// TIA Portal project "Event_Report" (V21)

(* hardware
DEVICE "S7-1200 station_1"  S7-1200 Station
   slot 0: "Rack_0"  S7-1200 Rack  Rack  V1.0
   slot 1: "PLC_1"  CPU 1215C AC/DC/Rly  6ES7 215-1BG40-0XB0  V4.2
*)

// ===== PLC "PLC_1"  CPU 1215C AC/DC/Rly =====

TYPE "UDT_CommBuffer"
VERSION : 0.1
   STRUCT
      SendTrigger : Bool;
      SendBuffer : Array[0..1023] of Byte;
      RecvBuffer : Array[0..1023] of Byte;
      RecvLength : UInt;
      RecvReady : Bool;
   END_STRUCT;
END_TYPE

DATA_BLOCK "DB_InputMonitor"   // DB1
{ S7_Optimized_Access := 'TRUE' }
VERSION : 0.1
   VAR
      InputImage : Array[1..100] of DWord;
      InputImage_Old : Array[1..100] of DWord;
      bSending : Bool;
   END_VAR
BEGIN
END_DATA_BLOCK

DATA_BLOCK "DB_CommData"   // DB3
{ S7_Optimized_Access := 'TRUE' }
AUTHOR : SIMATIC
VERSION : 0.1
   VAR
      SendLength : UInt;
      RecvLength : UInt;
      SendBuffer : Array[0..255] of Byte;
      RecvBuffer : Array[0..255] of Byte;
      StatusWord : Word;
   END_VAR
BEGIN
END_DATA_BLOCK

DATA_BLOCK "IDB_UdpTx"   // DB5
{ S7_Optimized_Access := 'TRUE' }
VERSION : 0.1
// stored: InstanceOfName FB_UdpTx
"FB_UdpTx"
BEGIN
END_DATA_BLOCK

DATA_BLOCK "IDB_MapDBtoIO"   // DB6
{ S7_Optimized_Access := 'TRUE' }
VERSION : 0.1
// stored: InstanceOfName FB_MapDBtoIO
"FB_MapDBtoIO"
BEGIN
   enable := true;
   tgtByte := 2;
   srcDB := 10;
   srcEndByte := 27;
   area := 16#81;
END_DATA_BLOCK

DATA_BLOCK "DB_input"   // DB10
{ S7_Optimized_Access := 'FALSE' }
VERSION : 0.1
   VAR
      "1层上行召梯按钮" : Bool;
      "2层上行召梯按钮" : Bool;
      "3层上行召梯按钮" : Bool;
      "4层上行召梯按钮" : Bool;
      "5层上行召梯按钮" : Bool;
      "6层上行召梯按钮" : Bool;
      "7层上行召梯按钮" : Bool;
      "8层上行召梯按钮" : Bool;
      "9层上行召梯按钮" : Bool;
      "2层下行召梯按钮" : Bool;
      "3层下行召梯按钮" : Bool;
      "4层下行召梯按钮" : Bool;
      "5层下行召梯按钮" : Bool;
      "6层下行召梯按钮" : Bool;
      "7层下行召梯按钮" : Bool;
      "8层下行召梯按钮" : Bool;
      "9层下行召梯按钮" : Bool;
      "10层下行召梯按钮" : Bool;
      "1号桥轿内选层按钮1" : Bool;
      "1号桥轿内选层按钮2" : Bool;
      "1号桥轿内选层按钮3" : Bool;
      "1号桥轿内选层按钮4" : Bool;
      "1号桥轿内选层按钮5" : Bool;
      "1号桥轿内选层按钮6" : Bool;
      "1号桥轿内选层按钮7" : Bool;
      "1号桥轿内选层按钮8" : Bool;
      "1号桥轿内选层按钮9" : Bool;
      "1号桥轿内选层按钮10" : Bool;
      "1号桥轿内开门按钮" : Bool;
      "1号桥轿内关门按钮" : Bool;
      "1号桥光幕信号" : Bool;
      "1号桥超重信号" : Bool;
      "1号桥检修信号" : Bool;
      "1号桥轿厢门门锁信号" : Bool;
      "1号桥1楼层门门锁信号" : Bool;
      "1号桥2楼层门门锁信号" : Bool;
      "1号桥3楼层门门锁信号" : Bool;
      "1号桥4楼层门门锁信号" : Bool;
      "1号桥5楼层门门锁信号" : Bool;
      "1号桥6楼层门门锁信号" : Bool;
      "1号桥7楼层门门锁信号" : Bool;
      "1号桥8楼层门门锁信号" : Bool;
      "1号桥9楼层门门锁信号" : Bool;
      "1号桥10楼层门门锁信号" : Bool;
      "1号桥开门到位" : Bool;
      "1号桥关门到位" : Bool;
      "1号桥上平层信号" : Bool;
      "1号桥下平层信号" : Bool;
      "1号桥上端站第1限位" : Bool;
      "1号桥上端站第2限位" : Bool;
      "1号桥下端站第1限位" : Bool;
      "1号桥下端站第2限位" : Bool;
      "2号桥轿内选层按钮1" : Bool;
      "2号桥轿内选层按钮2" : Bool;
      "2号桥轿内选层按钮3" : Bool;
      "2号桥轿内选层按钮4" : Bool;
      "2号桥轿内选层按钮5" : Bool;
      "2号桥轿内选层按钮6" : Bool;
      "2号桥轿内选层按钮7" : Bool;
      "2号桥轿内选层按钮8" : Bool;
      "2号桥轿内选层按钮9" : Bool;
      "2号桥轿内选层按钮10" : Bool;
      "2号桥轿内开门按钮" : Bool;
      "2号桥轿内关门按钮" : Bool;
      "2号桥光幕信号" : Bool;
      "2号桥超重信号" : Bool;
      "2号桥检修信号" : Bool;
      "2号桥轿厢门门锁信号" : Bool;
      "2号桥1楼层门门锁信号" : Bool;
      "2号桥2楼层门门锁信号" : Bool;
      "2号桥3楼层门门锁信号" : Bool;
      "2号桥4楼层门门锁信号" : Bool;
      "2号桥5楼层门门锁信号" : Bool;
      "2号桥6楼层门门锁信号" : Bool;
      "2号桥7楼层门门锁信号" : Bool;
      "2号桥8楼层门门锁信号" : Bool;
      "2号桥9楼层门门锁信号" : Bool;
      "2号桥10楼层门门锁信号" : Bool;
      "2号桥开门到位" : Bool;
      "2号桥关门到位" : Bool;
      "2号桥上平层信号" : Bool;
      "2号桥下平层信号" : Bool;
      "2号桥上端站第1限位" : Bool;
      "2号桥上端站第2限位" : Bool;
      "2号桥下端站第1限位" : Bool;
      "2号桥下端站第2限位" : Bool;
      "3号桥轿内选层按钮1" : Bool;
      "3号桥轿内选层按钮2" : Bool;
      "3号桥轿内选层按钮3" : Bool;
      "3号桥轿内选层按钮4" : Bool;
      "3号桥轿内选层按钮5" : Bool;
      "3号桥轿内选层按钮6" : Bool;
      "3号桥轿内选层按钮7" : Bool;
      "3号桥轿内选层按钮8" : Bool;
      "3号桥轿内选层按钮9" : Bool;
      "3号桥轿内选层按钮10" : Bool;
      "3号桥轿内开门按钮" : Bool;
      "3号桥轿内关门按钮" : Bool;
      "3号桥光幕信号" : Bool;
      "3号桥超重信号" : Bool;
      "3号桥检修信号" : Bool;
      "3号桥轿厢门门锁信号" : Bool;
      "3号桥1楼层门门锁信号" : Bool;
      "3号桥2楼层门门锁信号" : Bool;
      "3号桥3楼层门门锁信号" : Bool;
      "3号桥4楼层门门锁信号" : Bool;
      "3号桥5楼层门门锁信号" : Bool;
      "3号桥6楼层门门锁信号" : Bool;
      "3号桥7楼层门门锁信号" : Bool;
      "3号桥8楼层门门锁信号" : Bool;
      "3号桥9楼层门门锁信号" : Bool;
      "3号桥10楼层门门锁信号" : Bool;
      "3号桥开门到位" : Bool;
      "3号桥关门到位" : Bool;
      "3号桥上平层信号" : Bool;
      "3号桥下平层信号" : Bool;
      "3号桥上端站第1限位" : Bool;
      "3号桥上端站第2限位" : Bool;
      "3号桥下端站第1限位" : Bool;
      "3号桥下端站第2限位" : Bool;
      "4号桥轿内选层按钮1" : Bool;
      "4号桥轿内选层按钮2" : Bool;
      "4号桥轿内选层按钮3" : Bool;
      "4号桥轿内选层按钮4" : Bool;
      "4号桥轿内选层按钮5" : Bool;
      "4号桥轿内选层按钮6" : Bool;
      "4号桥轿内选层按钮7" : Bool;
      "4号桥轿内选层按钮8" : Bool;
      "4号桥轿内选层按钮9" : Bool;
      "4号桥轿内选层按钮10" : Bool;
      "4号桥轿内开门按钮" : Bool;
      "4号桥轿内关门按钮" : Bool;
      "4号桥光幕信号" : Bool;
      "4号桥超重信号" : Bool;
      "4号桥检修信号" : Bool;
      "4号桥轿厢门门锁信号" : Bool;
      "4号桥1楼层门门锁信号" : Bool;
      "4号桥2楼层门门锁信号" : Bool;
      "4号桥3楼层门门锁信号" : Bool;
      "4号桥4楼层门门锁信号" : Bool;
      "4号桥5楼层门门锁信号" : Bool;
      "4号桥6楼层门门锁信号" : Bool;
      "4号桥7楼层门门锁信号" : Bool;
      "4号桥8楼层门门锁信号" : Bool;
      "4号桥9楼层门门锁信号" : Bool;
      "4号桥10楼层门门锁信号" : Bool;
      "4号桥开门到位" : Bool;
      "4号桥关门到位" : Bool;
      "4号桥上平层信号" : Bool;
      "4号桥下平层信号" : Bool;
      "4号桥上端站第1限位" : Bool;
      "4号桥上端站第2限位" : Bool;
      "4号桥下端站第1限位" : Bool;
      "4号桥下端站第2限位" : Bool;
      "5号桥轿内选层按钮1" : Bool;
      "5号桥轿内选层按钮2" : Bool;
      "5号桥轿内选层按钮3" : Bool;
      "5号桥轿内选层按钮4" : Bool;
      "5号桥轿内选层按钮5" : Bool;
      "5号桥轿内选层按钮6" : Bool;
      "5号桥轿内选层按钮7" : Bool;
      "5号桥轿内选层按钮8" : Bool;
      "5号桥轿内选层按钮9" : Bool;
      "5号桥轿内选层按钮10" : Bool;
      "5号桥轿内开门按钮" : Bool;
      "5号桥轿内关门按钮" : Bool;
      "5号桥光幕信号" : Bool;
      "5号桥超重信号" : Bool;
      "5号桥检修信号" : Bool;
      "5号桥轿厢门门锁信号" : Bool;
      "5号桥1楼层门门锁信号" : Bool;
      "5号桥2楼层门门锁信号" : Bool;
      "5号桥3楼层门门锁信号" : Bool;
      "5号桥4楼层门门锁信号" : Bool;
      "5号桥5楼层门门锁信号" : Bool;
      "5号桥6楼层门门锁信号" : Bool;
      "5号桥7楼层门门锁信号" : Bool;
      "5号桥8楼层门门锁信号" : Bool;
      "5号桥9楼层门门锁信号" : Bool;
      "5号桥10楼层门门锁信号" : Bool;
      "5号桥开门到位" : Bool;
      "5号桥关门到位" : Bool;
      "5号桥上平层信号" : Bool;
      "5号桥下平层信号" : Bool;
      "5号桥上端站第1限位" : Bool;
      "5号桥上端站第2限位" : Bool;
      "5号桥下端站第1限位" : Bool;
      "5号桥下端站第2限位" : Bool;
      "6号桥轿内选层按钮1" : Bool;
      "6号桥轿内选层按钮2" : Bool;
      "6号桥轿内选层按钮3" : Bool;
      "6号桥轿内选层按钮4" : Bool;
      "6号桥轿内选层按钮5" : Bool;
      "6号桥轿内选层按钮6" : Bool;
      "6号桥轿内选层按钮7" : Bool;
      "6号桥轿内选层按钮8" : Bool;
      "6号桥轿内选层按钮9" : Bool;
      "6号桥轿内选层按钮10" : Bool;
      "6号桥轿内开门按钮" : Bool;
      "6号桥轿内关门按钮" : Bool;
      "6号桥光幕信号" : Bool;
      "6号桥超重信号" : Bool;
      "6号桥检修信号" : Bool;
      "6号桥轿厢门门锁信号" : Bool;
      "6号桥1楼层门门锁信号" : Bool;
      "6号桥2楼层门门锁信号" : Bool;
      "6号桥3楼层门门锁信号" : Bool;
      "6号桥4楼层门门锁信号" : Bool;
      "6号桥5楼层门门锁信号" : Bool;
      "6号桥6楼层门门锁信号" : Bool;
      "6号桥7楼层门门锁信号" : Bool;
      "6号桥8楼层门门锁信号" : Bool;
      "6号桥9楼层门门锁信号" : Bool;
      "6号桥10楼层门门锁信号" : Bool;
      "6号桥开门到位" : Bool;
      "6号桥关门到位" : Bool;
      "6号桥上平层信号" : Bool;
      "6号桥下平层信号" : Bool;
      "6号桥上端站第1限位" : Bool;
      "6号桥上端站第2限位" : Bool;
      "6号桥下端站第1限位" : Bool;
      "6号桥下端站第2限位" : Bool;
      自动运行信号 : Bool;
   END_VAR
BEGIN
END_DATA_BLOCK

DATA_BLOCK "DB_output"   // DB11
{ S7_Optimized_Access := 'FALSE' }
VERSION : 0.1
   VAR
      "1" : Bool;
      "2" : Bool;
      "3" : Bool;
      "4" : Bool;
      "5" : Bool;
      "6" : Bool;
      "7" : Bool;
      "8" : Bool;
      "9" : Bool;
      "10" : Bool;
      "11" : Bool;
      "12" : Bool;
      "13" : Bool;
      "14" : Bool;
      "15" : Bool;
      "16" : Bool;
      "17" : Bool;
      "18" : Bool;
      "19" : Bool;
      "20" : Bool;
      "21" : Bool;
      "22" : Bool;
      "23" : Bool;
      "24" : Bool;
      "25" : Bool;
      "26" : Bool;
      "27" : Bool;
      "28" : Bool;
      "29" : Bool;
      "30" : Bool;
      "31" : Bool;
      "32" : Bool;
      "33" : Bool;
      "34" : Bool;
      "35" : Bool;
      "36" : Bool;
      "37" : Bool;
      "38" : Bool;
      "39" : Bool;
      "40" : Bool;
      "41" : Bool;
      "42" : Bool;
      "43" : Bool;
      "44" : Bool;
      "45" : Bool;
      "46" : Bool;
      "47" : Bool;
      "48" : Bool;
      "49" : Bool;
      "50" : Bool;
      "51" : Bool;
      "52" : Bool;
      "53" : Bool;
      "54" : Bool;
      "55" : Bool;
      "56" : Bool;
      "57" : Bool;
      "58" : Bool;
      "59" : Bool;
      "60" : Bool;
      "61" : Bool;
      "62" : Bool;
      "63" : Bool;
      "64" : Bool;
      "65" : Bool;
      "66" : Bool;
      "67" : Bool;
      "68" : Bool;
      "69" : Bool;
      "70" : Bool;
      "71" : Bool;
      "72" : Bool;
      "73" : Bool;
      "74" : Bool;
      "75" : Bool;
      "76" : Bool;
      "77" : Bool;
      "78" : Bool;
      "79" : Bool;
      "80" : Bool;
      "81" : Bool;
      "82" : Bool;
      "83" : Bool;
      "84" : Bool;
      "85" : Bool;
      "86" : Bool;
      "87" : Bool;
      "88" : Bool;
      "89" : Bool;
      "90" : Bool;
      "91" : Bool;
      "92" : Bool;
      "93" : Bool;
      "94" : Bool;
      "95" : Bool;
      "96" : Bool;
      "97" : Bool;
      "98" : Bool;
      "99" : Bool;
      "100" : Bool;
      "101" : Bool;
      "102" : Bool;
      "103" : Bool;
      "104" : Bool;
      "105" : Bool;
      "106" : Bool;
      "107" : Bool;
      "108" : Bool;
      "109" : Bool;
      "110" : Bool;
      "111" : Bool;
      "112" : Bool;
      "113" : Bool;
      "114" : Bool;
      "115" : Bool;
      "116" : Bool;
      "117" : Bool;
      "118" : Bool;
      "119" : Bool;
      "120" : Bool;
      "121" : Bool;
      "122" : Bool;
      "123" : Bool;
      "124" : Bool;
      "125" : Bool;
      "126" : Bool;
      "127" : Bool;
      "128" : Bool;
      "129" : Bool;
      "130" : Bool;
      "131" : Bool;
      "132" : Bool;
      "133" : Bool;
      "134" : Bool;
      "135" : Bool;
      "136" : Bool;
      "137" : Bool;
      "138" : Bool;
      "139" : Bool;
      "140" : Bool;
      "141" : Bool;
      "142" : Bool;
      "143" : Bool;
      "144" : Bool;
      "145" : Bool;
      "146" : Bool;
      "147" : Bool;
      "148" : Bool;
      "149" : Bool;
      "150" : Bool;
      "151" : Bool;
      "152" : Bool;
      "153" : Bool;
      "154" : Bool;
      "155" : Bool;
      "156" : Bool;
      "157" : Bool;
      "158" : Bool;
      "159" : Bool;
      "160" : Bool;
      "161" : Bool;
      "162" : Bool;
      "163" : Bool;
      "164" : Bool;
      "165" : Bool;
      "166" : Bool;
      "167" : Bool;
      "168" : Bool;
      "169" : Bool;
      "170" : Bool;
      "171" : Bool;
      "172" : Bool;
      "173" : Bool;
      "174" : Bool;
      "175" : Bool;
      "176" : Bool;
      "177" : Bool;
      "178" : Bool;
      "179" : Bool;
      "180" : Bool;
      "181" : Bool;
      "182" : Bool;
      "183" : Bool;
      "184" : Bool;
      "185" : Bool;
      "186" : Bool;
      "187" : Bool;
      "188" : Bool;
      "189" : Bool;
      "190" : Bool;
      "191" : Bool;
      "192" : Bool;
      "193" : Bool;
      "194" : Bool;
      "195" : Bool;
      "196" : Bool;
      "197" : Bool;
      "198" : Bool;
      "199" : Bool;
      "200" : Bool;
      "201" : Bool;
      "202" : Bool;
      "203" : Bool;
      "204" : Bool;
      "205" : Bool;
      "206" : Bool;
      "207" : Bool;
      "208" : Bool;
      "209" : Bool;
      "210" : Bool;
      "211" : Bool;
      "212" : Bool;
      "213" : Bool;
      "214" : Bool;
      "215" : Bool;
      "216" : Bool;
      "217" : Bool;
      "218" : Bool;
      "219" : Bool;
      "220" : Bool;
      "221" : Bool;
      "222" : Bool;
      "223" : Bool;
      "224" : Bool;
      "225" : Bool;
      "226" : Bool;
      "227" : Bool;
      "228" : Bool;
      "229" : Bool;
      "230" : Bool;
      "231" : Bool;
      "232" : Bool;
      "233" : Bool;
      "234" : Bool;
      "235" : Bool;
      "236" : Bool;
      "237" : Bool;
      "238" : Bool;
      "239" : Bool;
      "240" : Bool;
      "241" : Bool;
      "242" : Bool;
      "243" : Bool;
      "244" : Bool;
      "245" : Bool;
      "246" : Bool;
      "247" : Bool;
      "248" : Bool;
      "249" : Bool;
      "250" : Bool;
      "251" : Bool;
      "252" : Bool;
      "253" : Bool;
      "254" : Bool;
      "255" : Bool;
      "256" : Bool;
      "257" : Bool;
      "258" : Bool;
      "259" : Bool;
      "260" : Bool;
      "261" : Bool;
      "262" : Bool;
      "263" : Bool;
      "264" : Bool;
   END_VAR
BEGIN
END_DATA_BLOCK

// folder: System blocks/Program resources

DATA_BLOCK "DB_TCON_Param"   // DB2
{ S7_Optimized_Access := 'TRUE' }
AUTHOR : SIMATIC
FAMILY : MC7Plus
NAME : TCON_Prm
VERSION : 1.0
// stored: InstanceOfName TCON_Param
"TCON_Param"
BEGIN
   ID := 1;
   LOCAL_TSAP_ID_LEN := 2;
   LOCAL_TSAP_ID[1] := 16#07;
   LOCAL_TSAP_ID[2] := 16#D0;
   REM_STADDR[1] := 192;
   REM_STADDR[2] := 168;
   REM_STADDR[3] := 1;
   REM_STADDR[4] := 201;
   REM_TSAP_ID[1] := 16#2C;
   REM_TSAP_ID[2] := 16#BB;
   CONNECTION_TYPE := 19;
   ACTIVE_EST := false;
END_DATA_BLOCK

// folder: (top level)

FUNCTION_BLOCK "FB_MapDBtoIO"   // FB1, SCL
{ S7_Optimized_Access := 'TRUE' }
VERSION : 0.1
   VAR_OUTPUT
      mappedBytes : Int;
      targetEndByte : Int;
   END_VAR
   VAR
      enable : Bool;
      tgtByte : Int;
      tgtBit : Int;
      srcDB : Int;
      srcByte : Int;
      srcEndByte : Int;
      area : Int;
      areaDB : Int;
   END_VAR
   VAR_TEMP
      i : Int;
      totalBits : Int;
      "b" : Bool;
      curByte : Int;
      curBit : Int;
      tByte : Int;
      tBit : Int;
   END_VAR
BEGIN
   // 计算映射字节数与目标结束字节
   #mappedBytes := #srcEndByte - #srcByte + 1;
   #targetEndByte := #tgtByte + #mappedBytes - 1;
   IF #tgtBit > 0 THEN
       #targetEndByte := #targetEndByte + 1;
   END_IF;

   IF #enable THEN
       #totalBits := #mappedBytes * 8 - 1;
       FOR #i := 0 TO #totalBits DO
           #curByte := #srcByte + #i / 8;
           #curBit  := #i MOD 8;
           #b := PEEK_BOOL(area := 16#84, dbNumber := #srcDB, byteOffset := #curByte, bitOffset := #curBit);
           #tByte := #tgtByte + (#tgtBit + #i) / 8;
           #tBit  := (#tgtBit + #i) MOD 8;
           POKE_BOOL(area := #area, dbNumber := #areaDB, byteOffset := #tByte, bitOffset := #tBit, value := #b);
       END_FOR;
   END_IF;
END_FUNCTION_BLOCK

FUNCTION_BLOCK "FB_UdpTx"   // FB2, SCL
{ S7_Optimized_Access := 'TRUE' }
VERSION : 0.1
   VAR_INPUT
      SendData : Bool;
   END_VAR
   VAR_OUTPUT
      SendDone : Bool;
      SendBusy : Bool;
      SendError : Bool;
      SendStatus : Word;
      UdpReady : Bool;
   END_VAR
   VAR
      tconInst : TCON;
      tusendInst : TUSEND;
      tconEdge : Bool;
      tconMem : Bool;
      tusendEdge : Bool;
      tusendMem : Bool;
      tconDone : Bool;
      tconBusy : Bool;
      tconErr : Bool;
      tconStat : Word;
      tusendDone : Bool;
      tusendBusy : Bool;
      tusendErr : Bool;
      tusendStat : Word;
      udpBound : Bool;
      remoteAddr : TADDR_Param;
      addrInit : Bool;
   END_VAR
BEGIN
   // Init remote address once
   IF NOT #addrInit THEN
       #remoteAddr.REM_IP_ADDR[1] := 192;
       #remoteAddr.REM_IP_ADDR[2] := 168;
       #remoteAddr.REM_IP_ADDR[3] := 1;
       #remoteAddr.REM_IP_ADDR[4] := 201;
       #remoteAddr.REM_PORT_NR := 11451;
       #addrInit := TRUE;
   END_IF;

   // TCON: bind UDP socket
   #tconEdge := NOT #udpBound AND NOT #tconMem;
   #tconMem := NOT #udpBound;
   #tconInst(REQ := #tconEdge,
             ID := 1,
             CONNECT := "DB_TCON_Param",
             DONE => #tconDone,
             BUSY => #tconBusy,
             ERROR => #tconErr,
             STATUS => #tconStat);
   IF #tconDone THEN
       #udpBound := TRUE;
   END_IF;
   IF #tconErr THEN
       #tconMem := FALSE;
   END_IF;

   // TUSEND: fire and forget
   // InputImage[1..25] = 100 bytes, 保持原 LEN=100 兼容旧接收端
   #tusendEdge := #SendData AND #udpBound AND NOT #tusendMem;
   #tusendMem := #SendData;
   #tusendInst(REQ := #tusendEdge,
               ID := 1,
               LEN := 100,
               DATA := "DB_CommData".SendBuffer,
               ADDR := #remoteAddr,
               DONE => #tusendDone,
               BUSY => #tusendBusy,
               ERROR => #tusendErr,
               STATUS => #tusendStat);

   #SendDone := #tusendDone;
   #SendBusy := #tusendBusy;
   #SendError := #tusendErr;
   #SendStatus := #tusendStat;
   #UdpReady := #udpBound;
END_FUNCTION_BLOCK

ORGANIZATION_BLOCK "OB100"   // OB1, SCL, ProgramCycle
TITLE = "Main Program Sweep (Cycle)"
{ S7_Optimized_Access := 'TRUE' }
VERSION : 0.1
   VAR_INPUT
      Initial_Call : Bool;   // Initial call of this OB
      Remanence : Bool;   // =True, if remanent data are available
   END_VAR
   VAR_TEMP
      i : Int;
   END_VAR
BEGIN
   FOR #i := 1 TO 100 DO
       "DB_InputMonitor".InputImage[#i] := 0;
   END_FOR;
END_ORGANIZATION_BLOCK

ORGANIZATION_BLOCK "Main"   // OB1, SCL, ProgramCycle
TITLE = "Main Program Sweep (Cycle)"
{ S7_Optimized_Access := 'TRUE' }
VERSION : 0.1
   VAR_INPUT
      Initial_Call : Bool;   // Initial call of this OB
      Remanence : Bool;   // =True, if remanent data are available
   END_VAR
   VAR_TEMP
      i : Int;
      dwTemp : DWord;
      j : Int;
      idx : Int;
      dwInp : DWord;
      bChanged : Bool;
      mapBytes : Int;
      targetEndByte : Int;
      readStart : Int;
      readIdx : Int;
   END_VAR
BEGIN
   // 0: 动态映射 DB10 → I 区（参数在 IDB_MapDBtoIO 在线设置）
   "IDB_MapDBtoIO"();
   #mapBytes := "IDB_MapDBtoIO".mappedBytes;
   #targetEndByte := "IDB_MapDBtoIO".targetEndByte;

   // 1: 清零 InputImage
   FOR #i := 1 TO 25 DO
       "DB_InputMonitor".InputImage[#i] := 0;
   END_FOR;

   // 2: 读物理 I0~I1 → InputImage[1] 低 2 字节
   #dwTemp := PEEK(area := 16#81, dbNumber := 0, byteOffset := 0);
   #dwTemp := #dwTemp AND 16#0000FFFF;
   "DB_InputMonitor".InputImage[1] := #dwTemp;

   // 3: 读映射区 I2~I3 → InputImage[1] 高 2 字节
   IF #targetEndByte >= 2 THEN
       #dwTemp := PEEK(area := 16#81, dbNumber := 0, byteOffset := 2);
       "DB_InputMonitor".InputImage[1] := "DB_InputMonitor".InputImage[1] OR SHL(IN := #dwTemp, N := 16);
   END_IF;

   // 4: 读映射区 I4~I7 → InputImage[2]
   IF #targetEndByte >= 4 THEN
       #dwTemp := PEEK(area := 16#81, dbNumber := 0, byteOffset := 4);
       "DB_InputMonitor".InputImage[2] := #dwTemp;
   END_IF;

   // 5: 读扩展映射区 I8~I29 → InputImage[3..8]
   #readStart := 8;
   #readIdx := 3;
   WHILE (#readStart <= #targetEndByte) AND (#readIdx <= 25) DO
       #dwTemp := PEEK(area := 16#81, dbNumber := 0, byteOffset := #readStart);
       "DB_InputMonitor".InputImage[#readIdx] := #dwTemp;
       #readStart := #readStart + 4;
       #readIdx := #readIdx + 1;
   END_WHILE;

   // 6: 检测变化
   #bChanged := FALSE;
   FOR #i := 1 TO 25 DO
       IF "DB_InputMonitor".InputImage[#i] <> "DB_InputMonitor".InputImage_Old[#i] THEN
           #bChanged := TRUE;
       END_IF;
   END_FOR;

   // 7: 有变化 → 打包到 SendBuffer
   IF #bChanged AND NOT "DB_InputMonitor".bSending THEN
       "DB_InputMonitor".bSending := TRUE;
       FOR #j := 1 TO 25 DO
           #dwInp := "DB_InputMonitor".InputImage[#j];
           #idx := (#j - 1) * 4;
           "DB_CommData".SendBuffer[#idx]    := DWORD_TO_BYTE(#dwInp);
           "DB_CommData".SendBuffer[#idx + 1] := DWORD_TO_BYTE(SHR(IN := #dwInp, N := 8));
           "DB_CommData".SendBuffer[#idx + 2] := DWORD_TO_BYTE(SHR(IN := #dwInp, N := 16));
           "DB_CommData".SendBuffer[#idx + 3] := DWORD_TO_BYTE(SHR(IN := #dwInp, N := 24));
       END_FOR;
       FOR #i := 1 TO 25 DO
           "DB_InputMonitor".InputImage_Old[#i] := "DB_InputMonitor".InputImage[#i];
       END_FOR;
   END_IF;

   // 8: UDP 发送完成或出错 → 清 bSending
   // 修复：原来只检查 SendDone，TUSEND 一次错误就导致 bSending 永久卡死
   IF "DB_InputMonitor".bSending AND ("IDB_UdpTx".SendDone OR "IDB_UdpTx".SendError) THEN
       "DB_InputMonitor".bSending := FALSE;
   END_IF;

   // 9: 触发 UDP 发送
   "IDB_UdpTx"(SendData := "DB_InputMonitor".bSending);
END_ORGANIZATION_BLOCK